FUNCTION_BLOCK FB_Peer (*EXTENDS FB_ComponentBase*) IMPLEMENTS I_Peer
VAR_INPUT
END_VAR
VAR_OUTPUT
END_VAR
VAR
	ePeer : E_PeersList;
	stMailbox : ST_Mailbox; 
END_VAR

PROPERTY eSetPeerId : E_PeersList
SET
ePeer := eSetPeerId;
END_SET
END_PROPERTY

METHOD M_CompareMessage : E_PeerReturnCode
VAR_INPUT
	in_stMessage : ST_Message;
END_VAR
VAR
	stIncomingMessage : ST_MESSAGE;
END_VAR
IF M_IsNewMessageAvailable() THEN
	
	stIncomingMessage := M_GetNextMessage();
	IF 	stIncomingMessage.eMessage = in_stMessage.eMessage
		AND stIncomingMessage.ePeer = in_stMessage.ePeer
		THEN
		
		M_CompareMessage := E_PeerReturnCode.eMATCH_FOUND;
		
	ELSE
		
		M_CompareMessage := E_PeerReturnCode.eNO_MATCH_FOUND;
	
	END_IF
	
ELSE

	M_CompareMessage := E_PeerReturnCode.eNO_NEW_MESSAGE;	
	
END_IF
END_METHOD

METHOD M_CompareMessageAndEmptyMailbox : E_PeerReturnCode
VAR_INPUT
	in_stMessage : ST_Message;
END_VAR
VAR
	stMessage : ST_Message;
	eTmpEval : E_PeerReturnCode;
END_VAR
M_CompareMessageAndEmptyMailbox := M_CompareMessage(in_stMessage);

IF M_CompareMessageAndEmptyMailbox = E_PeerReturnCode.eNO_MATCH_FOUND THEN
	stMessage := M_GetNextMessage();
	stMessage.eDeliveryStatus := E_DeliveryStatus.eDELIVERY_REJECTED;
	eTmpEval := M_SendMessage(stMessage);
END_IF

IF eTmpEval = E_PeerReturnCode.eMESSAGE_IN_OUTBOX
	OR M_CompareMessageAndEmptyMailbox = E_PeerReturnCode.eMATCH_FOUND
	THEN
	
	M_EmptyMailbox();
	
END_IF
END_METHOD

METHOD M_EmptyMailbox : E_PeerReturnCode
VAR_INPUT
END_VAR
VAR
	stEmptyMessage : ST_MESSAGE;
END_VAR
IF M_IsNewMessageAvailable() THEN
	stMailbox.stInbox := stEmptyMessage;
	stMailbox.bNewMessageAvail := FALSE;
	M_EmptyMailbox := E_PeerReturnCode.eMAILBOX_EMPTIED;
ELSE
	M_EmptyMailbox := E_PeerReturnCode.eMAILBOX_EMPTY;
END_IF
END_METHOD

METHOD M_GetNextMessage : ST_Message
IF M_IsNewMessageAvailable() THEN
	M_GetNextMessage := stMailbox.stInbox;
END_IF
END_METHOD

METHOD M_GetPeerId : E_PeersList
M_GetPeerId := ePeer;
END_METHOD

METHOD M_IsNewMessageAvailable : BOOL
M_IsNewMessageAvailable := stMailbox.bNewMessageAvail;
END_METHOD

METHOD M_RetrieveMailbox : REFERENCE TO ST_MAILBOX
VAR_INPUT
END_VAR
M_RetrieveMailbox Ref= stMailbox;
END_METHOD

METHOD M_SendMessage : E_PeerReturnCode
VAR_INPUT
	in_stMessage : ST_Message;
END_VAR
IF NOT stMailbox.bSendingMessage THEN
	stMailbox.stOutbox := in_stMessage;
	stMailbox.bSendingMessage := TRUE;
	M_SendMessage := E_PeerReturnCode.eMESSAGE_IN_OUTBOX;
ELSE
	M_SendMessage := E_PeerReturnCode.eMAILBOX_BUSY;
END_IF
END_METHOD

END_FUNCTION_BLOCK

(* stored: Version 1.1.0.1, ProductVersion 3.1.4022.12
   POU FB_Peer: Id {649f05f2-f8f7-4321-84e7-57ddb4422002}, SpecialFunc None
   Property eSetPeerId: Id {41b5b2fc-a03d-4a36-a554-b02e7f9b0db9}
   Set Set: Id {4c32e556-d653-41d4-9954-77a9f537d7d4}
   Method M_CompareMessage: Id {9acb8617-8d40-4e7e-9da3-0d06c79d32f3}
   Method M_CompareMessageAndEmptyMailbox: Id {d50a66b7-9de1-48fd-9e2f-1b5b2de39108}
   Method M_EmptyMailbox: Id {1c6fa322-ecc4-4159-893f-c6de54065be6}
   Method M_GetNextMessage: Id {83928553-9561-4ffa-9203-9059398e325b}
   Method M_GetPeerId: Id {a6b6b1ad-0a9b-4a1b-8a9b-b2bdb48762e5}
   Method M_IsNewMessageAvailable: Id {83d764a1-c7d8-4eeb-a4b4-2c8f522c9d72}
   Method M_RetrieveMailbox: Id {3aa7f8d2-d58a-46de-8339-a24562604a5d}
   Method M_SendMessage: Id {36db4a39-18fa-4cfd-b577-bb1450175a0f} *)
